# EPICS substitutions: BL03I-TEST/iocs/BL99I-LCH-IOC-01/BL99I-LCH-IOC-01App/Db/BL99I-LCH-IOC-01_expanded.substitutions
# This file was automatically generated on Wed 31 Oct 2018 13:49:07 GMT from
# source: /home/jjc62351/work/Builder/BL03I-TEST/etc/makeIocs/BL99I-LCH-IOC-01.xml
#
# *** Please do not edit this file: edit the source file instead. ***
#

# Macros:
#  IOC  Device prefix
file $(DEVIOCSTATS)/db/iocAdminVxWorks.db
{
pattern { IOC }
    { "BL22I-MO-IOC-03" }
}

# Macros:
#  IOC  Device prefix
file $(DEVIOCSTATS)/db/iocAdminScanMon.db
{
pattern { IOC }
    { "BL22I-MO-IOC-03" }
}

# Macros:
#  name      name for gui elements
#  EDM_FILE  edm screen, defaults to ioc_stats_softdls.edl
#  IOC       ioc name
file $(DEVIOCSTATS)/db/iocGui.db
{
pattern { name, EDM_FILE, IOC }
    { "IOCS.MO3", "ioc_stats_softdls.edl", "BL22I-MO-IOC-03" }
}

# Macros:
#  device  Device name
#  high    Temperature for MINOR severity alarm, default 50 deg
#  hihi    Temperature for MAJOR severity alarm, default 60 deg
#  hyst    Alarm deadband value, default 2 deg
file $(IOCINFO)/db/IOCinfo.template
{
pattern { device, high, hihi, hyst }
    { "BL22I-MO-IOC-03", "50", "60", "2" }
}

# Macros:
#  P        Device Prefix
#  PID      Device suffix
#  INP      Input PV for readback
#  OUT      Output PV for demand
#  SCAN     Scan rate for updating values on screen
#  KP       Proportional term for PID
#  KI       Integral term for PID
#  KD       Differential term for PID
#  LOPR     Low operating range of setopint
#  HOPR     High operating range of setopint
#  DRVL     Low limit on Output
#  DRVH     High limit on Output
#  PREC     Precision of display
#  AUTOPV   Shutter PV 1 to monitor to disable the PID
#  AUTOPV2  Shutter PV 2 to monitor to disable the PID
#  name     Object and gui association name
#  TITLE    Title of the EDM screen
file $(BLFEEDBACK)/db/feedback.template
{
pattern { P, PID, INP, OUT, SCAN, KP, KI, KD, LOPR, HOPR, DRVL, DRVH, PREC, AUTOPV, AUTOPV2, name, TITLE }
    { "BL22I-OP-DCM-01:FPMTR", ":FBS2", "BL22I-AL-SLITS-02:YPOS:FB PP NMS", "BL22I-OP-DCM-01:FPMTR:POUT", ".1 second", "1000", "0", "0", "-1000000", "1000000", "-10", "10", "7", "FE22I-RS-ABSB-02:STA", "BL22I-PS-SHTR-01:STA", "DCM.FEEDBACK", "Feedback" }
}

# Macros:
#  P         PV Prefix
#  Q         PV Suffix
#  DTYP      DTYP of bo records, e.g. Hy8001 or Soft Channel
#  OUTAC     Output link for AC/DC coupling bit, e.g. <RIOPV> PP
#  CAC       Card for AC/DC coupling bit, e.g. 70
#  SAC       Signal for AC/DC coupling bit, e.g. 35
#  gda_name  GDA name for amplifier, e.g. D1.AMP
file $(FEMTO)/db/femto_acdc200.template
{
pattern { P, Q, DTYP, OUTAC, CAC, SAC, gda_name }
    { "BL22I-DI-IAMP-10", "", "Hy8001", "#C$(CAC=) S$(SAC=) @", "100", "35", "" }
    { "BL22I-DI-IAMP-15", "", "Hy8001", "#C$(CAC=) S$(SAC=) @", "50", "35", "" }
    { "BL22I-DI-IAMP-16", "", "Hy8001", "#C$(CAC=) S$(SAC=) @", "50", "40", "" }
    { "BL22I-DI-IAMP-17", "", "Hy8001", "#C$(CAC=) S$(SAC=) @", "50", "45", "" }
    { "BL22I-DI-IAMP-18", "", "Hy8001", "#C$(CAC=) S$(SAC=) @", "100", "61", "" }
    { "BL22I-DI-IAMP-12", "", "Hy8001", "#C$(CAC=) S$(SAC=) @", "100", "45", "" }
    { "BL22I-DI-IAMP-13", "", "Hy8001", "#C$(CAC=) S$(SAC=) @", "100", "51", "" }
    { "BL22I-DI-PHDGN-04:BACKUP", ":DIODE2:AMP", "Hy8001", "#C$(CAC=) S$(SAC=) @", "50", "51", "" }
    { "BL22I-DI-PHDGN-06:BACKUP", ":DIODE2:AMP", "Hy8001", "#C$(CAC=) S$(SAC=) @", "50", "56", "" }
    { "BL22I-DI-PHDGN-04:BACKUP", ":DIODE1:AMP", "Hy8001", "#C$(CAC=) S$(SAC=) @", "100", "40", "" }
    { "BL22I-DI-PHDGN-06:BACKUP", ":DIODE1:AMP", "Hy8001", "#C$(CAC=) S$(SAC=) @", "100", "56", "" }
}

# Macros:
#  P         PV Prefix
#  Q         PV Suffix
#  INITGAIN  Initial gain value, e.g. 0
#  DTYP      DTYP of bo records, e.g. Hy8001 or Soft Channel
#  OUTGB0    Output link for gain bit 0, e.g. <RIOPV> PP
#  CGB0      Card for gain bit 0, e.g. 70
#  SGB0      Signal for gain bit 0, e.g. 32
#  OUTGB1    Output link for gain bit 1, e.g. <RIOPV> PP
#  CGB1      Card for gain bit 1, e.g. 70
#  SGB1      Signal for gain bit 1, e.g. 33
#  OUTGB2    Output link for gain bit 2, e.g. <RIOPV> PP
#  CGB2      Card for gain bit 2, e.g. 70
#  SGB2      Signal for gain bit 2, e.g. 34
#  OUTHIS    Output link for High speed/Low noise bit, e.g. <RIOPV> PP
#  CHIS      Card for High speed/Low noise bit, e.g. 70
#  SHIS      Signal for High speed/Low noise bit, e.g. 36
#  gda_name  GDA name for amplifier, e.g. D1.AMP
#  gda_desc  GDA description for name for amplifier, e.g. D1.AMP
#  name      Object and gui association name
file $(FEMTO)/db/femto200.template
{
pattern { P, Q, INITGAIN, DTYP, OUTGB0, CGB0, SGB0, OUTGB1, CGB1, SGB1, OUTGB2, CGB2, SGB2, OUTHIS, CHIS, SHIS, gda_name, gda_desc, name }
    { "BL22I-AL-SLITS-02", ":YMDRAIN", "0", "Hy8001", "#C$(CGB0=) S$(SGB0=) @", "100", "42", "#C$(CGB1=) S$(SGB1=) @", "100", "43", "#C$(CGB2=) S$(SGB2=) @", "100", "44", "#C$(CHIS=) S$(SHIS=) @", "100", "46", "IAMP12CTR", "Current amp12 control", "S2.YMAMP" }
    { "BL22I-AL-SLITS-02", ":YPDRAIN", "0", "Hy8001", "#C$(CGB0=) S$(SGB0=) @", "100", "48", "#C$(CGB1=) S$(SGB1=) @", "100", "49", "#C$(CGB2=) S$(SGB2=) @", "100", "50", "#C$(CHIS=) S$(SHIS=) @", "100", "52", "IAMP13CTR", "Current amp13 control", "S2.YPAMP" }
    { "BL22I-DI-PHDGN-04:BACKUP", ":DIODE1", "0", "Hy8001", "#C$(CGB0=) S$(SGB0=) @", "100", "37", "#C$(CGB1=) S$(SGB1=) @", "100", "38", "#C$(CGB2=) S$(SGB2=) @", "100", "39", "#C$(CHIS=) S$(SHIS=) @", "100", "41", "D4I1", "D4 Diode 1 femto", "D4.D1AMP" }
    { "BL22I-DI-PHDGN-06:BACKUP", ":DIODE1", "0", "Hy8001", "#C$(CGB0=) S$(SGB0=) @", "100", "53", "#C$(CGB1=) S$(SGB1=) @", "100", "54", "#C$(CGB2=) S$(SGB2=) @", "100", "55", "#C$(CHIS=) S$(SHIS=) @", "100", "57", "D6I1", "D6 Diode 1 femto", "D6.D1AMP" }
    { "BL22I-DI-PHDGN-04:BACKUP", ":DIODE2", "0", "Hy8001", "#C$(CGB0=) S$(SGB0=) @", "50", "48", "#C$(CGB1=) S$(SGB1=) @", "50", "49", "#C$(CGB2=) S$(SGB2=) @", "50", "50", "#C$(CHIS=) S$(SHIS=) @", "50", "52", "D4I2", "D4 Diode 2 femto", "D4.D2AMP" }
    { "BL22I-DI-PHDGN-06:BACKUP", ":DIODE2", "0", "Hy8001", "#C$(CGB0=) S$(SGB0=) @", "50", "53", "#C$(CGB1=) S$(SGB1=) @", "50", "54", "#C$(CGB2=) S$(SGB2=) @", "50", "55", "#C$(CHIS=) S$(SHIS=) @", "50", "57", "D6I2", "D6 Diode 2 femto", "D6.D2AMP" }
}

# Macros:
#  P         PV Prefix
#  Q         PV Suffix, should probably end in :I
#  DESC      Description
#  DTYPE     DTYP of record, e.g. asynInt32
#  INP       Input link of record, e.g. @asyn(ADC1 0) GENDATA
#  EGU       Engineering units
#  EGUF      EGUs full scale
#  EGUL      EGUs low scale
#  SCAN      Scan rate
#  PREC      Precision
#  HOPR      High operating range
#  LOPR      High operating range
#  ADEL      Alarm deadband
#  gda_name  GDA name for amplifier, e.g. D1.AMP
file $(FEMTO)/db/femto_ai.template
{
pattern { P, Q, DESC, DTYPE, INP, EGU, EGUF, EGUL, SCAN, PREC, HOPR, LOPR, ADEL, gda_name }
    { "BL22I-DI-PHDGN-04:BACKUP", ":DIODE2:I", "D4 current 2", "asynFloat64", "@asyn(ADC90 7) GENDATA", "", "10", "-10", "I/O Intr", "3", "10", "-10", "0.002", "D4I2" }
}

# Macros:
#  P  Template argument
#  Q  Template argument
file $(ELETTRASY900S)/db/elettraSY900Sbimorph.template
{
pattern { P, Q }
    { "BL22I-OP-KBM-01", ":VFM" }
    { "BL22I-OP-KBM-01", ":HFM" }
}

# Macros:
#  P         Template argument
#  Q         Template argument
#  gda_name  Template argument
#  gda_desc  Template argument
file $(ELETTRASY900S)/db/elettraSY900Sgda16.template
{
pattern { P, Q, gda_name, gda_desc }
    { "BL22I-OP-KBM-01", ":VFM", "VFMBIMORPH", "VFM bimorph" }
}

# Macros:
#  P         Template argument
#  Q         Template argument
#  gda_name  Template argument
#  gda_desc  Template argument
file $(ELETTRASY900S)/db/elettraSY900Sgda6.template
{
pattern { P, Q, gda_name, gda_desc }
    { "BL22I-OP-KBM-01", ":HFM", "HFMBIMORPH", "HFM bimorph" }
}

# Macros:
#  P         Device Prefix
#  R         Device Suffix
#  DTYP      Device Type
#  INP       Input link
#  SCAN      Scan Rate
#  ZNAM      Name for zero state
#  ONAM      Name for one state
#  ZSV       optional macro to allow zero state alarm severity to be set.
#  OSV       optional macro to allow one state alarm severity to be set.
#  COSV      optional macro to allow change of state alarm severity to be set.
#  DESC      Description
#  name      Object name and gui association name
#  gda_name  GDA Name
#  gda_desc  GDA Description
file $(USERIO)/db/bi.template
{
pattern { P, R, DTYP, INP, SCAN, ZNAM, ONAM, ZSV, OSV, COSV, DESC, name, gda_name, gda_desc }
    { "BL22I-OP-KBM-01:UPS", "", "Hy8001", "#C40 S39 @", "1 second", "UPS", "MAINS", "", "", "", "Binary Input", "IOCS.UPS", "KBM1UPS", "UPS detection" }
}

# Macros:
#  P         Device Prefix
#  R         Device Suffix
#  DTYP      Device Type
#  OUT       Output link
#  SCAN      Scan Rate
#  EGUL      EGU low scale
#  EGUF      EGU full scale
#  DRVH      Drive high limit
#  DRVL      Drive low limit
#  LINR      LINR
#  PREC      Precision
#  EGU       EGU
#  PINI      Process on iocInit
#  DESC      Description
#  name      Object name and gui association name
#  gda_name  GDA Name
#  gda_desc  GDA Description
file $(USERIO)/db/ao.template
{
pattern { P, R, DTYP, OUT, SCAN, EGUL, EGUF, DRVH, DRVL, LINR, PREC, EGU, PINI, DESC, name, gda_name, gda_desc }
    { "BL22I-OP-KBM-01", ":HFM:FY3:OUT", "asynInt32", "@asyn(DAC92, 0)", "Passive", "-10", "10", "10", "-10", "LINEAR", "", "V", "NO", "Analogue Output", "", "", "" }
    { "BL22I-OP-KBM-01", ":VFM:FY3:OUT", "asynInt32", "@asyn(DAC92, 1)", "Passive", "-10", "10", "10", "-10", "LINEAR", "", "V", "NO", "Analogue Output", "", "", "" }
}

# Macros:
#  P         Device Prefix
#  R         Device Suffix
#  DTYP      Device Type
#  INP       Input link
#  SCAN      Scan Rate
#  PREC      Precision
#  EGUL      EGU low scale
#  EGUF      EGU full scale
#  EGU       EGU
#  LINR      LINR
#  DESC      Description
#  name      Object name and gui association name
#  gda_name  GDA Name
#  gda_desc  GDA Description
file $(USERIO)/db/ai.template
{
pattern { P, R, DTYP, INP, SCAN, PREC, EGUL, EGUF, EGU, LINR, DESC, name, gda_name, gda_desc }
    { "BL22I-OP-KBM-01", ":HFM:FY3:RBV", "asynInt32", "@asyn(ADC90 5) GENDATA", "I/O Intr", "5", "-10", "10", "V", "LINEAR", "Analogue Input", "", "", "" }
    { "BL22I-OP-KBM-01", ":VFM:FY3:RBV", "asynInt32", "@asyn(ADC90 6) GENDATA", "I/O Intr", "5", "-10", "10", "V", "LINEAR", "Analogue Input", "", "", "" }
}

# Macros:
#  P         Device Prefix
#  Q         Device Suffix
#  DESC      Description, displayed on EDM screen
#  RDBL      Readback link
#  OUT       Output link
#  MOVEDLY   Approximate move time (seconds)
#  EGU       Engineering Units
#  DHLM      Dial High Limit
#  DLLM      Dial Low Limit
#  MRES      Motor Step Size (EGU)
#  RRES      Readback Step Size (EGU)
#  RDBD      Retry deadband (EGU)
#  name      Object name and gui association name
#  gda_name  Name to export this as to GDA
#  gda_desc  Description to export this as to GDA
file $(MOTOR)/db/softMotorForPiezo.template
{
pattern { P, Q, DESC, RDBL, OUT, MOVEDLY, EGU, DHLM, DLLM, MRES, RRES, RDBD, name, gda_name, gda_desc }
    { "BL22I-OP-KBM-01", ":HFM:FY3", "Fine horizontal", "BL22I-OP-KBM-01:HFM:FY3:RBV", "BL22I-OP-KBM-01:HFM:FY3:OUT", "0.25", "V", "10", "-10", "0.0001", "1", "0.0001", "HFM.FY3", "", "" }
    { "BL22I-OP-KBM-01", ":VFM:FY3", "Fine vertical", "BL22I-OP-KBM-01:VFM:FY3:RBV", "BL22I-OP-KBM-01:VFM:FY3:OUT", "0.25", "V", "10", "-10", "0.0001", "1", "0.0001", "VFM.FY3", "", "" }
}

# Macros:
#  P     Template argument
#  R     Template argument
#  PORT  Template argument
#  ADDR  Template argument
#  OMAX  Template argument
#  IMAX  Template argument
file $(ASYN)/db/asynRecord.db
{
pattern { P, R, PORT, ADDR, OMAX, IMAX }
    { "BL22I-MO-IOC-03", ":ASYN", "", "", "1024", "1024" }
}

# Macros:
#  device  Template argument
#  c       Template argument
#  s       Template argument
#  DTYP    Template argument
file $(RACKFAN)/db/rackFan.template
{
pattern { device, c, s, DTYP }
    { "BL22I-MO-FANC-01", "40", "32", "Hy8001" }
    { "BL22I-MO-FANC-02", "40", "33", "Hy8001" }
    { "BL22I-MO-FANC-03", "40", "34", "Hy8001" }
    { "BL22I-MO-FANC-04", "40", "36", "Hy8001" }
}

# Macros:
#  device      Template argument
#  BL_SECTION  Template argument
file $(CRYOCOOLER)/db/devCryocooler.template
{
pattern { device, BL_SECTION }
    { "BL22I-CG-CRYO-01", "ALL" }
}

# Macros:
#  device      Template argument
#  ALARM_NAME  Template argument
#  DESC        Template argument
#  DTYP        Template argument
#  ONAM        Template argument
#  ZNAM        Template argument
#  NUM         Template argument
file $(CRYOCOOLER)/db/devCryocoolerAlarm.template
{
pattern { device, ALARM_NAME, DESC, DTYP, ONAM, ZNAM, NUM }
    { "BL22I-CG-CRYO-01", "AL1", "Buff. N probe fault", "Cryocooler", "ON", "OFF", "30" }
    { "BL22I-CG-CRYO-01", "AL2", "Main vessel N probe fault", "Cryocooler", "ON", "OFF", "31" }
    { "BL22I-CG-CRYO-01", "AL3", "N feed pr. trans. fault", "Cryocooler", "ON", "OFF", "32" }
    { "BL22I-CG-CRYO-01", "AL4", "N return pr. trans. fault", "Cryocooler", "ON", "OFF", "33" }
    { "BL22I-CG-CRYO-01", "AL5", "Pump oper. curr. det. fault", "Cryocooler", "ON", "OFF", "34" }
    { "BL22I-CG-CRYO-01", "AL6", "N flow trans. fault", "Cryocooler", "ON", "OFF", "35" }
    { "BL22I-CG-CRYO-01", "AL7", "N feed temp. sensor fault", "Cryocooler", "ON", "OFF", "36" }
    { "BL22I-CG-CRYO-01", "AL8", "N return temp. sensor fault", "Cryocooler", "ON", "OFF", "37" }
    { "BL22I-CG-CRYO-01", "AL9", "Top plate temp. sensor fault", "Cryocooler", "ON", "OFF", "38" }
    { "BL22I-CG-CRYO-01", "AL10", "Objective temp. sensor fault", "Cryocooler", "ON", "OFF", "39" }
    { "BL22I-CG-CRYO-01", "AL11", "Spare", "Cryocooler", "ON", "OFF", "40" }
    { "BL22I-CG-CRYO-01", "AL12", "Spare", "Cryocooler", "ON", "OFF", "41" }
    { "BL22I-CG-CRYO-01", "AL13", "Int. 24V supply fuse blown", "Cryocooler", "ON", "OFF", "42" }
    { "BL22I-CG-CRYO-01", "AL14", "Ext. 24V supply fuse blown", "Cryocooler", "ON", "OFF", "43" }
    { "BL22I-CG-CRYO-01", "AL15", "Earth leakage break. tripped", "Cryocooler", "ON", "OFF", "44" }
    { "BL22I-CG-CRYO-01", "AL16", "Press. cont. heat. tripped", "Cryocooler", "ON", "OFF", "45" }
    { "BL22I-CG-CRYO-01", "AL17", "Anti condens. heat. tripped", "Cryocooler", "ON", "OFF", "46" }
    { "BL22I-CG-CRYO-01", "AL18", "Pump motor MCB tripped", "Cryocooler", "ON", "OFF", "47" }
    { "BL22I-CG-CRYO-01", "AL19", "Spare", "Cryocooler", "ON", "OFF", "48" }
    { "BL22I-CG-CRYO-01", "AL20", "Spare", "Cryocooler", "ON", "OFF", "49" }
    { "BL22I-CG-CRYO-01", "AL21", "N buff. press. below band", "Cryocooler", "ON", "OFF", "50" }
    { "BL22I-CG-CRYO-01", "AL22", "N buff. press above band", "Cryocooler", "ON", "OFF", "51" }
    { "BL22I-CG-CRYO-01", "AL23", "N buff. press trip", "Cryocooler", "ON", "OFF", "52" }
    { "BL22I-CG-CRYO-01", "AL24", "N feed press trip", "Cryocooler", "ON", "OFF", "53" }
    { "BL22I-CG-CRYO-01", "AL25", "N flow rate below band", "Cryocooler", "ON", "OFF", "54" }
    { "BL22I-CG-CRYO-01", "AL26", "N flow rate above band", "Cryocooler", "ON", "OFF", "55" }
    { "BL22I-CG-CRYO-01", "AL27", "N pump overcurrent alarm", "Cryocooler", "ON", "OFF", "56" }
    { "BL22I-CG-CRYO-01", "AL28", "Spare", "Cryocooler", "ON", "OFF", "57" }
    { "BL22I-CG-CRYO-01", "AL29", "Vessel N level low warning", "Cryocooler", "ON", "OFF", "58" }
    { "BL22I-CG-CRYO-01", "AL30", "Vessel N level low trip", "Cryocooler", "ON", "OFF", "59" }
    { "BL22I-CG-CRYO-01", "AL31", "Vessel N level high warning", "Cryocooler", "ON", "OFF", "60" }
    { "BL22I-CG-CRYO-01", "AL32", "Vessel N level high trip", "Cryocooler", "ON", "OFF", "61" }
    { "BL22I-CG-CRYO-01", "AL33", "Vessel N level over maximum", "Cryocooler", "ON", "OFF", "62" }
    { "BL22I-CG-CRYO-01", "AL34", "Buffer N level low trip", "Cryocooler", "ON", "OFF", "63" }
    { "BL22I-CG-CRYO-01", "AL35", "Buffer N level high warning", "Cryocooler", "ON", "OFF", "64" }
    { "BL22I-CG-CRYO-01", "AL36", "Buffer N level high trip", "Cryocooler", "ON", "OFF", "65" }
    { "BL22I-CG-CRYO-01", "AL37", "Pump on with low buff. level", "Cryocooler", "ON", "OFF", "66" }
    { "BL22I-CG-CRYO-01", "AL38", "Pump con. failed to engage", "Cryocooler", "ON", "OFF", "67" }
    { "BL22I-CG-CRYO-01", "AL39", "Pump contactor dropped out", "Cryocooler", "ON", "OFF", "68" }
    { "BL22I-CG-CRYO-01", "AL40", "No response from pump cont.", "Cryocooler", "ON", "OFF", "69" }
    { "BL22I-CG-CRYO-01", "AL41", "Pump controller tripped", "Cryocooler", "ON", "OFF", "70" }
    { "BL22I-CG-CRYO-01", "AL42", "Spare", "Cryocooler", "ON", "OFF", "71" }
    { "BL22I-CG-CRYO-01", "AL43", "Spare", "Cryocooler", "ON", "OFF", "72" }
    { "BL22I-CG-CRYO-01", "AL44", "Heat. cont. failed to engage", "Cryocooler", "ON", "OFF", "73" }
    { "BL22I-CG-CRYO-01", "AL45", "Heater cont. dropped out", "Cryocooler", "ON", "OFF", "74" }
    { "BL22I-CG-CRYO-01", "AL46", "Spare", "Cryocooler", "ON", "OFF", "75" }
    { "BL22I-CG-CRYO-01", "AL47", "Spare", "Cryocooler", "ON", "OFF", "76" }
    { "BL22I-CG-CRYO-01", "AL48", "Cryocooler restarted", "Cryocooler", "ON", "OFF", "77" }
    { "BL22I-CG-CRYO-01", "AL49", "Autofill diss. -> cryo. run.", "Cryocooler", "ON", "OFF", "78" }
    { "BL22I-CG-CRYO-01", "AL50", "Pump stopped -> cryo. run.", "Cryocooler", "ON", "OFF", "79" }
    { "BL22I-CG-CRYO-01", "AL51", "Press. cont. disabled wh", "Cryocooler", "ON", "OFF", "80" }
    { "BL22I-CG-CRYO-01", "AL52", "Spare", "Cryocooler", "ON", "OFF", "81" }
    { "BL22I-CG-CRYO-01", "AL53", "Spare", "Cryocooler", "ON", "OFF", "82" }
    { "BL22I-CG-CRYO-01", "AL54", "Spare", "Cryocooler", "ON", "OFF", "83" }
    { "BL22I-CG-CRYO-01", "AL55", "Spare", "Cryocooler", "ON", "OFF", "84" }
    { "BL22I-CG-CRYO-01", "AL56", "Spare", "Cryocooler", "ON", "OFF", "85" }
    { "BL22I-CG-CRYO-01", "AL57", "Spare", "Cryocooler", "ON", "OFF", "86" }
    { "BL22I-CG-CRYO-01", "AL58", "Spare", "Cryocooler", "ON", "OFF", "87" }
    { "BL22I-CG-CRYO-01", "AL59", "Spare", "Cryocooler", "ON", "OFF", "88" }
    { "BL22I-CG-CRYO-01", "AL60", "Spare", "Cryocooler", "ON", "OFF", "89" }
}
